// TIA Portal project "Project_ToggleButton_Sım" (V16)

(* hardware
DEVICE "S7-1200 station_1"  S7-1200 Station
   slot 0: "Rack_0"  S7-1200 Rack  Rack  V1.0
   slot 1: "PLC_1"  CPU 1212C DC/DC/Rly  6ES7 212-1HE40-0XB0  V4.4
*)

// ===== PLC "PLC_1"  CPU 1212C DC/DC/Rly =====

VAR_GLOBAL   // PLC tag table "Default tag table"
   ""TOGGLE BUTON"" AT %I0.0 : Bool;
   ""CIKIS"" AT %Q0.0 : Bool;
END_VAR